FUNCTION Convert_DINT_TO_LREAL : Hresult
VAR_INPUT
	in : DINT;
	out : REFERENCE TO LREAL;
END_VAR
VAR
	converted : LREAL;
END_VAR
VAR CONSTANT
	INCOMPATIBLE : HRESULT := 16#9811070E;
END_VAR

converted := DINT_TO_LREAL(in);

IF (LREAL_TO_DINT(converted) <> in) THEN
	Convert_DINT_TO_LREAL := INCOMPATIBLE;
	RETURN;
END_IF

out := converted;

END_FUNCTION

(* stored: Version 1.1.0.1, ProductVersion 3.1.4024.12
   POU Convert_DINT_TO_LREAL: Id {d390f6a3-c6f6-450b-a90e-66306280dcb8}, SpecialFunc None *)
